FUNCTION_BLOCK PAEPump EXTENDS PAEEMotor1D
VAR_INPUT
END_VAR
VAR_OUTPUT
END_VAR
VAR
END_VAR

END_FUNCTION_BLOCK

(* stored: Version 1.1.0.1, ProductVersion 3.1.4020.12
   POU PAEPump: Id {7a66110a-4a7e-46dc-9b32-a364f5508800}, SpecialFunc None *)
